
TYPE "DriveControlOutput"
STRUCT
        driveStatus : WORD;
        actualSpeed : INT;
END_STRUCT;
END_TYPE